Fanuc TP program (LS listing): MSG40.LS

/PROG  MSG40
/ATTR
OWNER		= MNEDITOR;
COMMENT		= "MESSAGE 40 chars";
PROG_SIZE	= 214;
CREATE		= DATE 26-09-18  TIME 15:08:28;
MODIFIED	= DATE 26-09-18  TIME 15:08:28;
FILE_NAME	= ;
VERSION		= 0;
LINE_COUNT	= 1;
MEMORY_SIZE	= 582;
PROTECT		= READ_WRITE;
TCD:  STACK_SIZE	= 0,
      TASK_PRIORITY	= 50,
      TIME_SLICE	= 0,
      BUSY_LAMP_OFF	= 0,
      ABORT_REQUEST	= 0,
      PAUSE_REQUEST	= 0;
DEFAULT_GROUP	= 1,*,*,*,*;
CONTROL_CODE	= 00000000 00000000;
LOCAL_REGISTERS	= 0,0,0;
/MN
   1:  MESSAGE[ABCDEFGHIJKLMNOPQRSTUVWX] ;
/POS
/END
